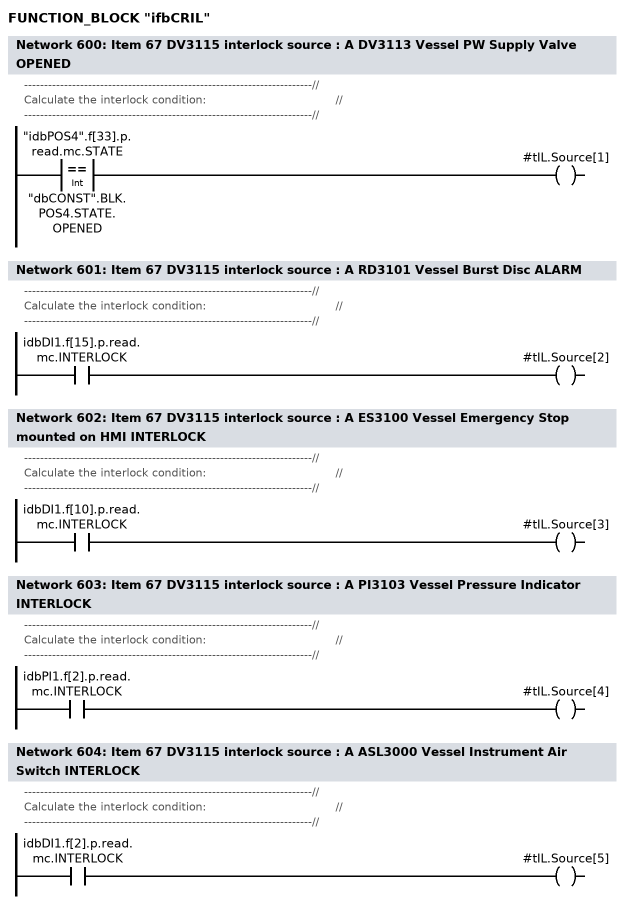
    A(;
    L "idbPOS4".f[33].p.read.mc.STATE;
    L "dbCONST".BLK.POS4.STATE.OPENED;
    ==I;
    );
    = #tIL.Source[1];

NETWORK
TITLE = Item 67 DV3115 interlock source : A RD3101 Vessel Burst Disc ALARM
    //------------------------------------------------------------------------//
    // Calculate the interlock condition:                                     //
    //------------------------------------------------------------------------//
    A idbDI1.f[15].p.read.mc.INTERLOCK;
    = #tIL.Source[2];

NETWORK
TITLE = Item 67 DV3115 interlock source : A ES3100 Vessel Emergency Stop mounted on HMI INTERLOCK
    //------------------------------------------------------------------------//
    // Calculate the interlock condition:                                     //
    //------------------------------------------------------------------------//
    A idbDI1.f[10].p.read.mc.INTERLOCK;
    = #tIL.Source[3];

NETWORK
TITLE = Item 67 DV3115 interlock source : A PI3103 Vessel Pressure Indicator INTERLOCK
    //------------------------------------------------------------------------//
    // Calculate the interlock condition:                                     //
    //------------------------------------------------------------------------//
    A idbPI1.f[2].p.read.mc.INTERLOCK;
    = #tIL.Source[4];

NETWORK
TITLE = Item 67 DV3115 interlock source : A ASL3000 Vessel Instrument Air Switch INTERLOCK
    //------------------------------------------------------------------------//
    // Calculate the interlock condition:                                     //
    //------------------------------------------------------------------------//
    A idbDI1.f[2].p.read.mc.INTERLOCK;
    = #tIL.Source[5];

NETWORK
TITLE = Item 67 DV3115 interlock source : AN ZSC3101 Vessel Manway Closed Indicator CLOSED
    //------------------------------------------------------------------------//
    // Calculate the interlock condition:                                     //
    //------------------------------------------------------------------------//
    AN(;
    L "idbZSC1".f[2].p.read.mc.STATE;
    L "dbCONST".BLK.ZSC1.STATE.CLOSED;
    ==I;
    );
    = #tIL.Source[6];


NETWORK
TITLE = Item 67 DV3115 : Number of interlocks
    //------------------------------------------------------------------------//
    // Number of interlocks
    //------------------------------------------------------------------------//
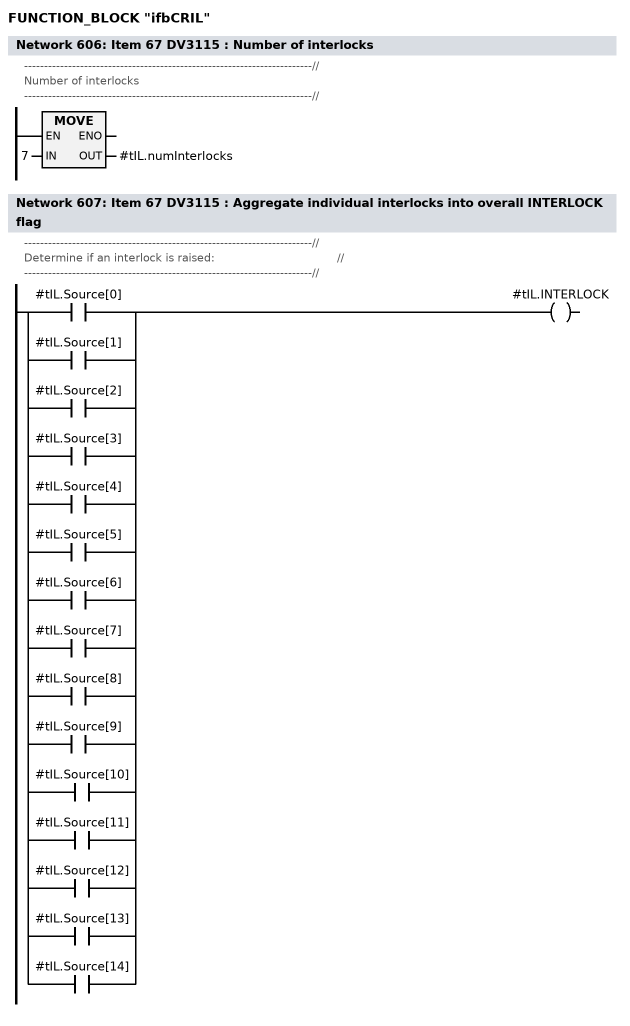
    L 7;
    T #tIL.numInterlocks;

NETWORK
TITLE = Item 67 DV3115 : Aggregate individual interlocks into overall INTERLOCK flag
    //------------------------------------------------------------------------//
    // Determine if an interlock is raised:                                   //
    //------------------------------------------------------------------------//
    O #tIL.Source[0];
    O #tIL.Source[1];
    O #tIL.Source[2];
    O #tIL.Source[3];
    O #tIL.Source[4];
    O #tIL.Source[5];
    O #tIL.Source[6];
    O #tIL.Source[7];
    O #tIL.Source[8];
    O #tIL.Source[9];
    O #tIL.Source[10];
    O #tIL.Source[11];
    O #tIL.Source[12];
    O #tIL.Source[13];
    O #tIL.Source[14];
    = #tIL.INTERLOCK;

NETWORK
TITLE = Item 67 DV3115 : Update the instance data
    //------------------------------------------------------------------------//
    // Update the instance DB with the calculated interlock flags:            //
    //------------------------------------------------------------------------//
    CALL MOVE
    {value_type := 'Variant'}
    (   IN                   := #tIL ,
        OUT                  := #p[67]
    );

NETWORK
TITLE = Item 68 DV3117 : Spray Ball 1 Valve initialise variables
    //------------------------------------------------------------------------//
    // CRITICAL INTERLOCK   CRITICAL INTERLOCK   CRITICAL INTERLOCK   CRITICA //
    // CRITICAL INTERLOCK   CRITICAL INTERLOCK   CRITICAL INTERLOCK   CRITICA //
    //                                                                        //
    // Clear the interlock flag:                                              //
    //------------------------------------------------------------------------//
    A "alwaysLow";
    = #tIL.INTERLOCK;

    //------------------------------------------------------------------------//
    // Clear all interlock values to initialise them to off:                  //
    //------------------------------------------------------------------------//
    CALL FILL_BLK
    {value_type := 'Bool', count_type := 'UInt'}
    (   IN                   := 0 ,
        COUNT                := 15 ,
        OUT                  := #tIL.Source[0]
    );


NETWORK
TITLE = Item 68 DV3117 interlock source : A RD3101 Vessel Burst Disc ALARM
    //------------------------------------------------------------------------//
    // Calculate the interlock condition:                                     //
    //------------------------------------------------------------------------//
    A idbDI1.f[15].p.read.mc.INTERLOCK;
    = #tIL.Source[0];

NETWORK
TITLE = Item 68 DV3117 interlock source : A ES3100 Vessel Emergency Stop mounted on HMI INTERLOCK
    //------------------------------------------------------------------------//
    // Calculate the interlock condition:                                     //
    //------------------------------------------------------------------------//
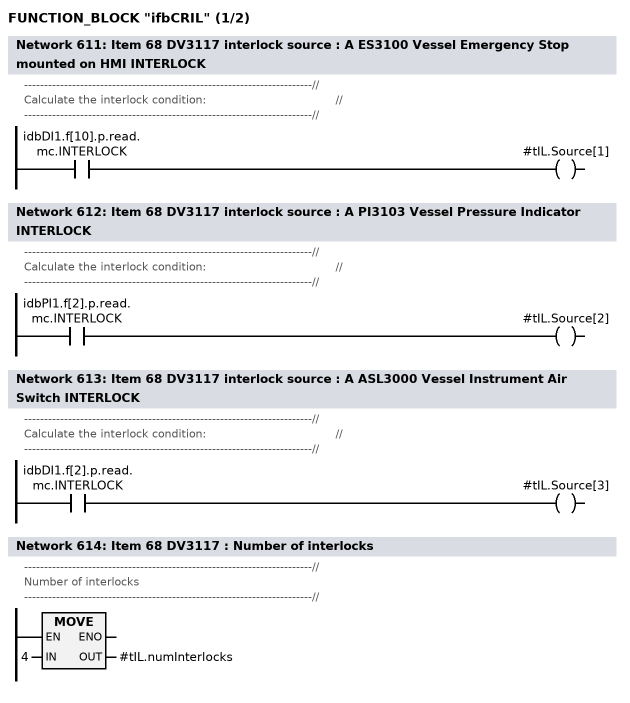
    A idbDI1.f[10].p.read.mc.INTERLOCK;
    = #tIL.Source[1];

NETWORK
TITLE = Item 68 DV3117 interlock source : A PI3103 Vessel Pressure Indicator INTERLOCK
    //------------------------------------------------------------------------//
    // Calculate the interlock condition:                                     //
    //------------------------------------------------------------------------//
    A idbPI1.f[2].p.read.mc.INTERLOCK;
    = #tIL.Source[2];

NETWORK
TITLE = Item 68 DV3117 interlock source : A ASL3000 Vessel Instrument Air Switch INTERLOCK
    //------------------------------------------------------------------------//
    // Calculate the interlock condition:                                     //
    //------------------------------------------------------------------------//
    A idbDI1.f[2].p.read.mc.INTERLOCK;
    = #tIL.Source[3];


NETWORK
TITLE = Item 68 DV3117 : Number of interlocks
    //------------------------------------------------------------------------//
    // Number of interlocks
    //------------------------------------------------------------------------//
    L 4;
    T #tIL.numInterlocks;

NETWORK
TITLE = Item 68 DV3117 : Aggregate individual interlocks into overall INTERLOCK flag
    //------------------------------------------------------------------------//
    // Determine if an interlock is raised:                                   //
    //------------------------------------------------------------------------//
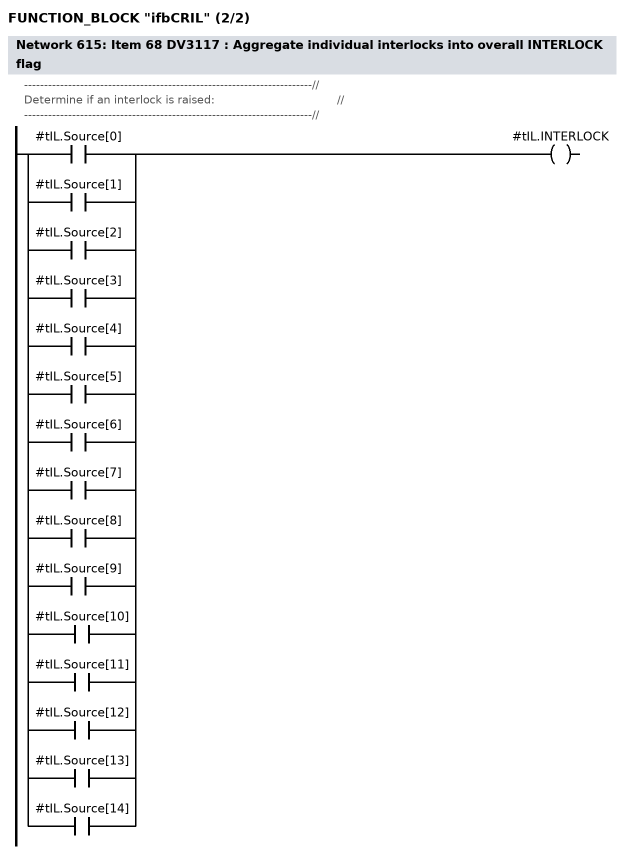
    O #tIL.Source[0];
    O #tIL.Source[1];
    O #tIL.Source[2];
    O #tIL.Source[3];
    O #tIL.Source[4];
    O #tIL.Source[5];
    O #tIL.Source[6];
    O #tIL.Source[7];
    O #tIL.Source[8];
    O #tIL.Source[9];
    O #tIL.Source[10];
    O #tIL.Source[11];
    O #tIL.Source[12];
    O #tIL.Source[13];
    O #tIL.Source[14];
    = #tIL.INTERLOCK;

NETWORK
TITLE = Item 68 DV3117 : Update the instance data
    //------------------------------------------------------------------------//
    // Update the instance DB with the calculated interlock flags:            //
    //------------------------------------------------------------------------//
    CALL MOVE
    {value_type := 'Variant'}
    (   IN                   := #tIL ,
        OUT                  := #p[68]
    );

NETWORK
TITLE = Item 69 DV3119 : Spray Ball 2 Valve initialise variables
    //------------------------------------------------------------------------//
    // CRITICAL INTERLOCK   CRITICAL INTERLOCK   CRITICAL INTERLOCK   CRITICA //
    // CRITICAL INTERLOCK   CRITICAL INTERLOCK   CRITICAL INTERLOCK   CRITICA //
    //                                                                        //
    // Clear the interlock flag:                                              //
    //------------------------------------------------------------------------//
    A "alwaysLow";
    = #tIL.INTERLOCK;

    //------------------------------------------------------------------------//
    // Clear all interlock values to initialise them to off:                  //
    //------------------------------------------------------------------------//
    CALL FILL_BLK
    {value_type := 'Bool', count_type := 'UInt'}
    (   IN                   := 0 ,
        COUNT                := 15 ,
        OUT                  := #tIL.Source[0]
    );


NETWORK
TITLE = Item 69 DV3119 interlock source : A RD3101 Vessel Burst Disc ALARM
    //------------------------------------------------------------------------//
    // Calculate the interlock condition:                                     //
    //------------------------------------------------------------------------//
    A idbDI1.f[15].p.read.mc.INTERLOCK;
    = #tIL.Source[0];

NETWORK
TITLE = Item 69 DV3119 interlock source : A ES3100 Vessel Emergency Stop mounted on HMI INTERLOCK
    //------------------------------------------------------------------------//
    // Calculate the interlock condition:                                     //
    //------------------------------------------------------------------------//
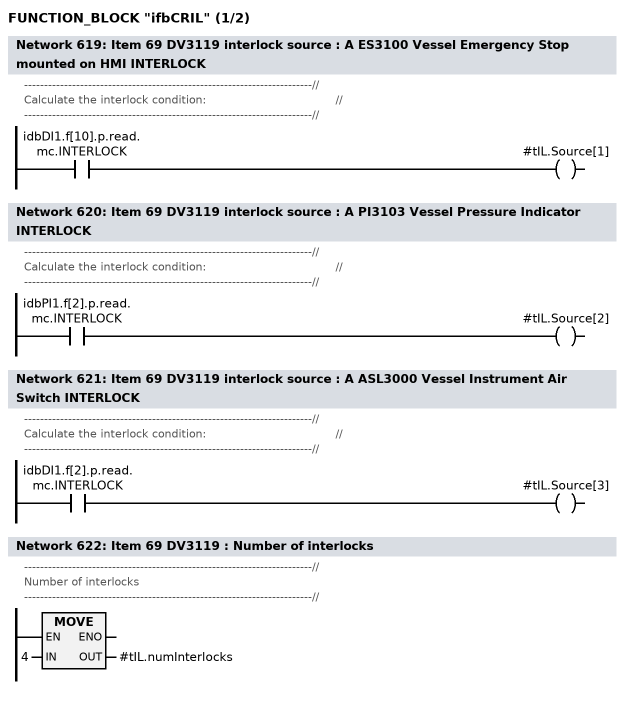
    A idbDI1.f[10].p.read.mc.INTERLOCK;
    = #tIL.Source[1];

NETWORK
TITLE = Item 69 DV3119 interlock source : A PI3103 Vessel Pressure Indicator INTERLOCK
    //------------------------------------------------------------------------//
    // Calculate the interlock condition:                                     //
    //------------------------------------------------------------------------//
    A idbPI1.f[2].p.read.mc.INTERLOCK;
    = #tIL.Source[2];

NETWORK
TITLE = Item 69 DV3119 interlock source : A ASL3000 Vessel Instrument Air Switch INTERLOCK
    //------------------------------------------------------------------------//
    // Calculate the interlock condition:                                     //
    //------------------------------------------------------------------------//
    A idbDI1.f[2].p.read.mc.INTERLOCK;
    = #tIL.Source[3];


NETWORK
TITLE = Item 69 DV3119 : Number of interlocks
    //------------------------------------------------------------------------//
    // Number of interlocks
    //------------------------------------------------------------------------//
    L 4;
    T #tIL.numInterlocks;

NETWORK
TITLE = Item 69 DV3119 : Aggregate individual interlocks into overall INTERLOCK flag
    //------------------------------------------------------------------------//
    // Determine if an interlock is raised:                                   //
    //------------------------------------------------------------------------//
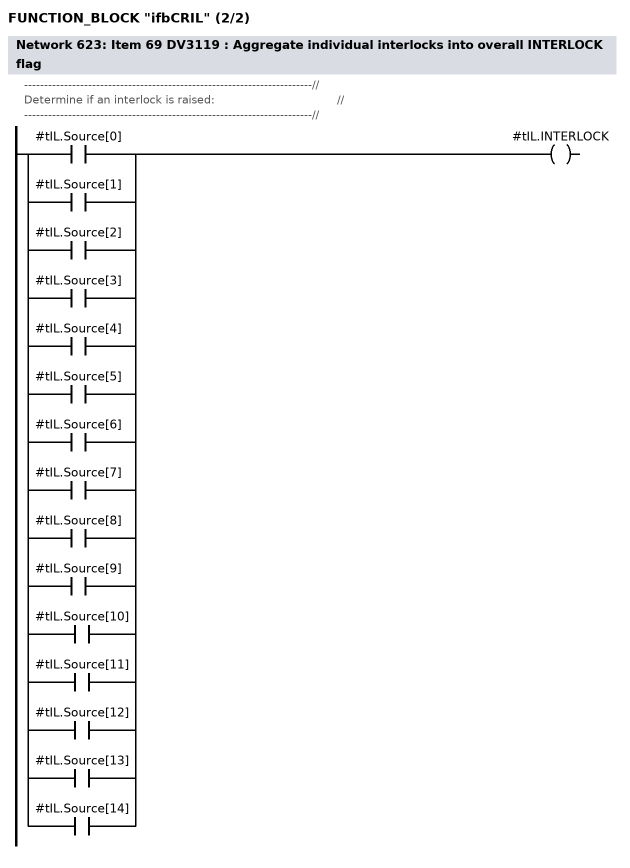
    O #tIL.Source[0];
    O #tIL.Source[1];
    O #tIL.Source[2];
    O #tIL.Source[3];
    O #tIL.Source[4];
    O #tIL.Source[5];
    O #tIL.Source[6];
    O #tIL.Source[7];
    O #tIL.Source[8];
    O #tIL.Source[9];
    O #tIL.Source[10];
    O #tIL.Source[11];
    O #tIL.Source[12];
    O #tIL.Source[13];
    O #tIL.Source[14];
    = #tIL.INTERLOCK;

NETWORK
TITLE = Item 69 DV3119 : Update the instance data
    //------------------------------------------------------------------------//
    // Update the instance DB with the calculated interlock flags:            //
    //------------------------------------------------------------------------//
    CALL MOVE
    {value_type := 'Variant'}
    (   IN                   := #tIL ,
        OUT                  := #p[69]
    );

NETWORK
TITLE = Item 70 DV3121 : Outlet Valve initialise variables
    //------------------------------------------------------------------------//
    // CRITICAL INTERLOCK   CRITICAL INTERLOCK   CRITICAL INTERLOCK   CRITICA //
    // CRITICAL INTERLOCK   CRITICAL INTERLOCK   CRITICAL INTERLOCK   CRITICA //
    //                                                                        //
    // Clear the interlock flag:                                              //
    //------------------------------------------------------------------------//
    A "alwaysLow";
    = #tIL.INTERLOCK;

    //------------------------------------------------------------------------//
    // Clear all interlock values to initialise them to off:                  //
    //------------------------------------------------------------------------//
    CALL FILL_BLK
    {value_type := 'Bool', count_type := 'UInt'}
    (   IN                   := 0 ,
        COUNT                := 15 ,
        OUT                  := #tIL.Source[0]
    );


NETWORK
TITLE = Item 70 DV3121 interlock source : A RD3101 Vessel Burst Disc ALARM
    //------------------------------------------------------------------------//
    // Calculate the interlock condition:                                     //
    //------------------------------------------------------------------------//
    A idbDI1.f[15].p.read.mc.INTERLOCK;
    = #tIL.Source[0];

NETWORK
TITLE = Item 70 DV3121 interlock source : A ES3100 Vessel Emergency Stop mounted on HMI INTERLOCK
    //------------------------------------------------------------------------//
    // Calculate the interlock condition:                                     //
    //------------------------------------------------------------------------//
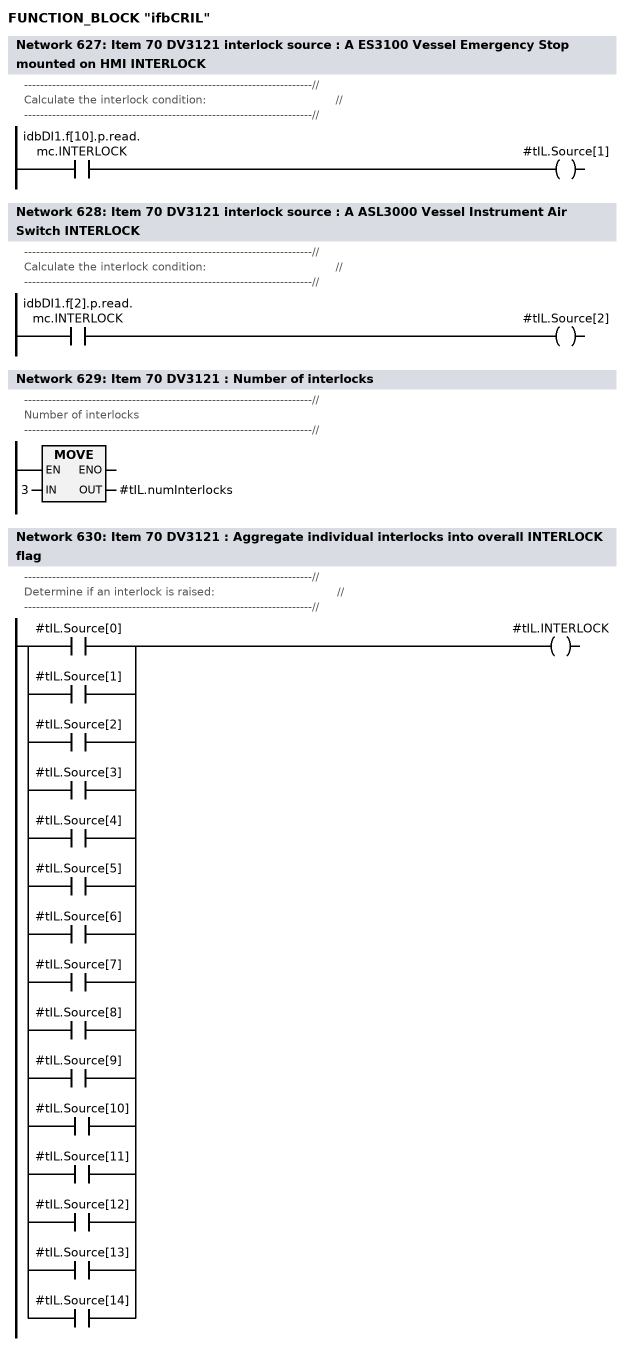
    A idbDI1.f[10].p.read.mc.INTERLOCK;
    = #tIL.Source[1];

NETWORK
TITLE = Item 70 DV3121 interlock source : A ASL3000 Vessel Instrument Air Switch INTERLOCK
    //------------------------------------------------------------------------//
    // Calculate the interlock condition:                                     //
    //------------------------------------------------------------------------//
    A idbDI1.f[2].p.read.mc.INTERLOCK;
    = #tIL.Source[2];


NETWORK
TITLE = Item 70 DV3121 : Number of interlocks
    //------------------------------------------------------------------------//
    // Number of interlocks
    //------------------------------------------------------------------------//
    L 3;
    T #tIL.numInterlocks;

NETWORK
TITLE = Item 70 DV3121 : Aggregate individual interlocks into overall INTERLOCK flag
    //------------------------------------------------------------------------//
    // Determine if an interlock is raised:                                   //
    //------------------------------------------------------------------------//
    O #tIL.Source[0];
    O #tIL.Source[1];
    O #tIL.Source[2];
    O #tIL.Source[3];
    O #tIL.Source[4];
    O #tIL.Source[5];
    O #tIL.Source[6];
    O #tIL.Source[7];
    O #tIL.Source[8];
    O #tIL.Source[9];
    O #tIL.Source[10];
    O #tIL.Source[11];
    O #tIL.Source[12];
    O #tIL.Source[13];
    O #tIL.Source[14];
    = #tIL.INTERLOCK;

NETWORK
TITLE = Item 70 DV3121 : Update the instance data
    //------------------------------------------------------------------------//
    // Update the instance DB with the calculated interlock flags:            //
    //------------------------------------------------------------------------//
    CALL MOVE
    {value_type := 'Variant'}
    (   IN                   := #tIL ,
        OUT                  := #p[70]
    );

NETWORK
TITLE = Item 71 DV3125 : Sy Transfer line Valve Matrix SMFLx initialise variables
    //------------------------------------------------------------------------//
    // CRITICAL INTERLOCK   CRITICAL INTERLOCK   CRITICAL INTERLOCK   CRITICA //
    // CRITICAL INTERLOCK   CRITICAL INTERLOCK   CRITICAL INTERLOCK   CRITICA //
    //                                                                        //
    // Clear the interlock flag:                                              //
    //------------------------------------------------------------------------//
    A "alwaysLow";
    = #tIL.INTERLOCK;

    //------------------------------------------------------------------------//
    // Clear all interlock values to initialise them to off:                  //
    //------------------------------------------------------------------------//
    CALL FILL_BLK
    {value_type := 'Bool', count_type := 'UInt'}
    (   IN                   := 0 ,
        COUNT                := 15 ,
        OUT                  := #tIL.Source[0]
    );


NETWORK
TITLE = Item 71 DV3125 interlock source : AN ZSC3111 SMFL1 to S1/BFS1 Flowpath Indicator IN   AN ZSC3113 SMFL2 to S1/BFS1 Flowpath Indicator IN
    //------------------------------------------------------------------------//
    // Calculate the interlock condition:                                     //
    //------------------------------------------------------------------------//
    AN(;
    L "idbZSC2".f[17].p.read.mc.STATE;
    L "dbCONST".BLK.ZSC2.STATE.IN;
    ==I;
    );
AN(;
    L "idbZSC2".f[18].p.read.mc.STATE;
    L "dbCONST".BLK.ZSC2.STATE.IN;
    ==I;
    );
    = #tIL.Source[0];


NETWORK
TITLE = Item 71 DV3125 : Number of interlocks
    //------------------------------------------------------------------------//
    // Number of interlocks
    //------------------------------------------------------------------------//
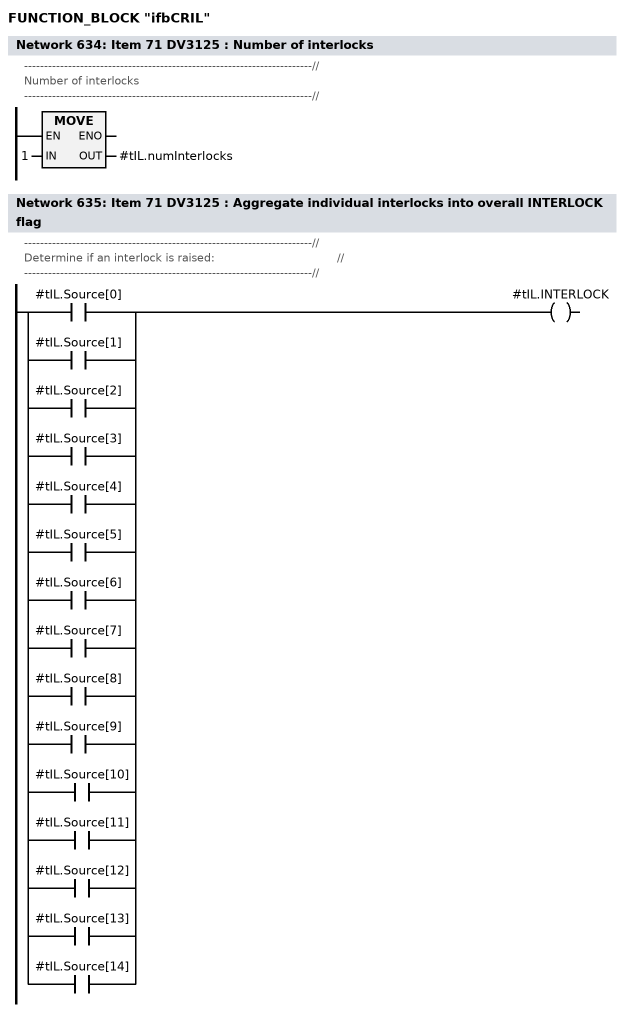
    L 1;
    T #tIL.numInterlocks;

NETWORK
TITLE = Item 71 DV3125 : Aggregate individual interlocks into overall INTERLOCK flag
    //------------------------------------------------------------------------//
    // Determine if an interlock is raised:                                   //
    //------------------------------------------------------------------------//
    O #tIL.Source[0];
    O #tIL.Source[1];
    O #tIL.Source[2];
    O #tIL.Source[3];
    O #tIL.Source[4];
    O #tIL.Source[5];
    O #tIL.Source[6];
    O #tIL.Source[7];
    O #tIL.Source[8];
    O #tIL.Source[9];
    O #tIL.Source[10];
    O #tIL.Source[11];
    O #tIL.Source[12];
    O #tIL.Source[13];
    O #tIL.Source[14];
    = #tIL.INTERLOCK;

NETWORK
TITLE = Item 71 DV3125 : Update the instance data
    //------------------------------------------------------------------------//
    // Update the instance DB with the calculated interlock flags:            //
    //------------------------------------------------------------------------//
    CALL MOVE
    {value_type := 'Variant'}
    (   IN                   := #tIL ,
        OUT                  := #p[71]
    );

NETWORK
TITLE = Item 72 DV3129 : Sy Transfer line Valve Matrix FLz initialise variables
    //------------------------------------------------------------------------//
    // CRITICAL INTERLOCK   CRITICAL INTERLOCK   CRITICAL INTERLOCK   CRITICA //
    // CRITICAL INTERLOCK   CRITICAL INTERLOCK   CRITICAL INTERLOCK   CRITICA //
    //                                                                        //
    // Clear the interlock flag:                                              //
    //------------------------------------------------------------------------//
    A "alwaysLow";
    = #tIL.INTERLOCK;

    //------------------------------------------------------------------------//
    // Clear all interlock values to initialise them to off:                  //
    //------------------------------------------------------------------------//
    CALL FILL_BLK
    {value_type := 'Bool', count_type := 'UInt'}
    (   IN                   := 0 ,
        COUNT                := 15 ,
        OUT                  := #tIL.Source[0]
    );


NETWORK
TITLE = Item 72 DV3129 interlock source : AN ZSC3115 S1 to F1P1 Flowpath Indicator IN   AN ZSC3117 S1 to F2P1 Flowpath Indicator IN
    //------------------------------------------------------------------------//
    // Calculate the interlock condition:                                     //
    //------------------------------------------------------------------------//
    AN(;
    L "idbZSC2".f[19].p.read.mc.STATE;
    L "dbCONST".BLK.ZSC2.STATE.IN;
    ==I;
    );
AN(;
    L "idbZSC2".f[20].p.read.mc.STATE;
    L "dbCONST".BLK.ZSC2.STATE.IN;
    ==I;
    );
    = #tIL.Source[0];


NETWORK
TITLE = Item 72 DV3129 : Number of interlocks
    //------------------------------------------------------------------------//
    // Number of interlocks
    //------------------------------------------------------------------------//
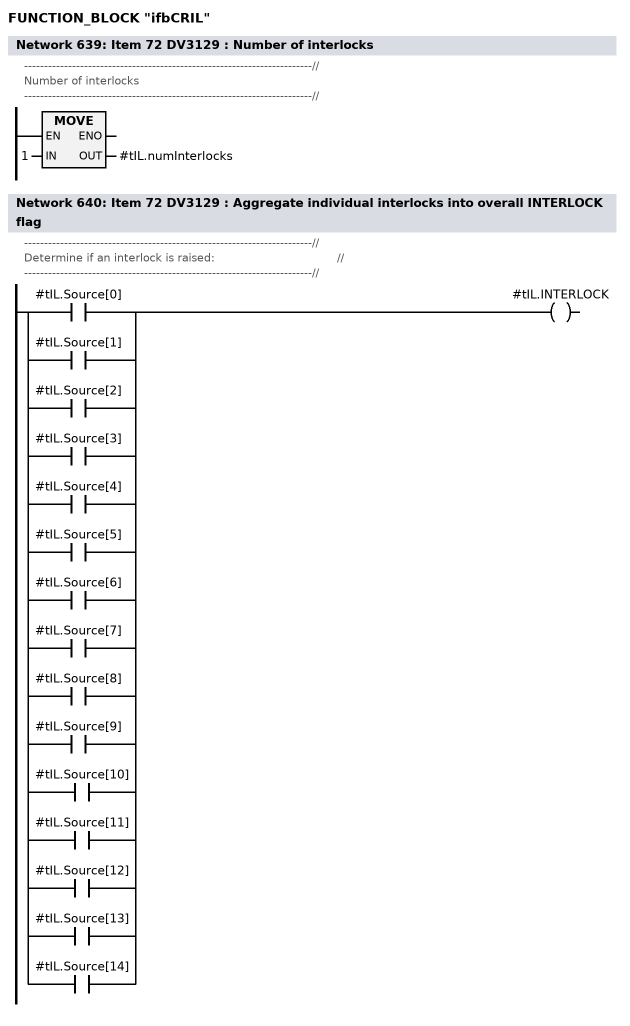
    L 1;
    T #tIL.numInterlocks;

NETWORK
TITLE = Item 72 DV3129 : Aggregate individual interlocks into overall INTERLOCK flag
    //------------------------------------------------------------------------//
    // Determine if an interlock is raised:                                   //
    //------------------------------------------------------------------------//
    O #tIL.Source[0];
    O #tIL.Source[1];
    O #tIL.Source[2];
    O #tIL.Source[3];
    O #tIL.Source[4];
    O #tIL.Source[5];
    O #tIL.Source[6];
    O #tIL.Source[7];
    O #tIL.Source[8];
    O #tIL.Source[9];
    O #tIL.Source[10];
    O #tIL.Source[11];
    O #tIL.Source[12];
    O #tIL.Source[13];
    O #tIL.Source[14];
    = #tIL.INTERLOCK;

NETWORK
TITLE = Item 72 DV3129 : Update the instance data
    //------------------------------------------------------------------------//
    // Update the instance DB with the calculated interlock flags:            //
    //------------------------------------------------------------------------//
    CALL MOVE
    {value_type := 'Variant'}
    (   IN                   := #tIL ,
        OUT                  := #p[72]
    );

NETWORK
TITLE = Item 73 DV4101 : Vent Valve initialise variables
    //------------------------------------------------------------------------//
    // CRITICAL INTERLOCK   CRITICAL INTERLOCK   CRITICAL INTERLOCK   CRITICA //
    // CRITICAL INTERLOCK   CRITICAL INTERLOCK   CRITICAL INTERLOCK   CRITICA //
    //                                                                        //
    // Clear the interlock flag:                                              //
    //------------------------------------------------------------------------//
    A "alwaysLow";
    = #tIL.INTERLOCK;

    //------------------------------------------------------------------------//
    // Clear all interlock values to initialise them to off:                  //
    //------------------------------------------------------------------------//
    CALL FILL_BLK
    {value_type := 'Bool', count_type := 'UInt'}
    (   IN                   := 0 ,
        COUNT                := 15 ,
        OUT                  := #tIL.Source[0]
    );


NETWORK
TITLE = Item 73 DV4101 interlock source : A RD4101 Vessel Burst Disc ALARM
    //------------------------------------------------------------------------//
    // Calculate the interlock condition:                                     //
    //------------------------------------------------------------------------//
    A idbDI1.f[16].p.read.mc.INTERLOCK;
    = #tIL.Source[0];

NETWORK
TITLE = Item 73 DV4101 interlock source : A ES4100 Vessel Emergency Stop mounted on HMI INTERLOCK
    //------------------------------------------------------------------------//
    // Calculate the interlock condition:                                     //
    //------------------------------------------------------------------------//
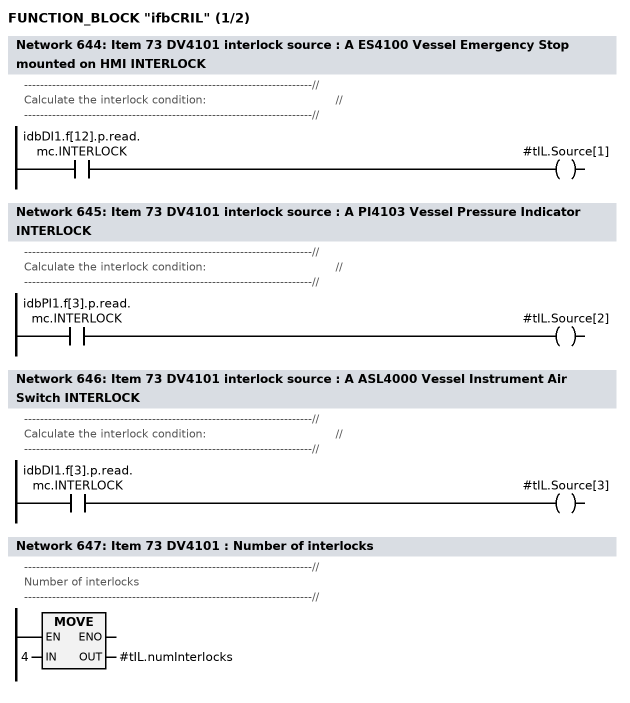
    A idbDI1.f[12].p.read.mc.INTERLOCK;
    = #tIL.Source[1];

NETWORK
TITLE = Item 73 DV4101 interlock source : A PI4103 Vessel Pressure Indicator INTERLOCK
    //------------------------------------------------------------------------//
    // Calculate the interlock condition:                                     //
    //------------------------------------------------------------------------//
    A idbPI1.f[3].p.read.mc.INTERLOCK;
    = #tIL.Source[2];

NETWORK
TITLE = Item 73 DV4101 interlock source : A ASL4000 Vessel Instrument Air Switch INTERLOCK
    //------------------------------------------------------------------------//
    // Calculate the interlock condition:                                     //
    //------------------------------------------------------------------------//
    A idbDI1.f[3].p.read.mc.INTERLOCK;
    = #tIL.Source[3];


NETWORK
TITLE = Item 73 DV4101 : Number of interlocks
    //------------------------------------------------------------------------//
    // Number of interlocks
    //------------------------------------------------------------------------//
    L 4;
    T #tIL.numInterlocks;

NETWORK
TITLE = Item 73 DV4101 : Aggregate individual interlocks into overall INTERLOCK flag
    //------------------------------------------------------------------------//
    // Determine if an interlock is raised:                                   //
    //------------------------------------------------------------------------//
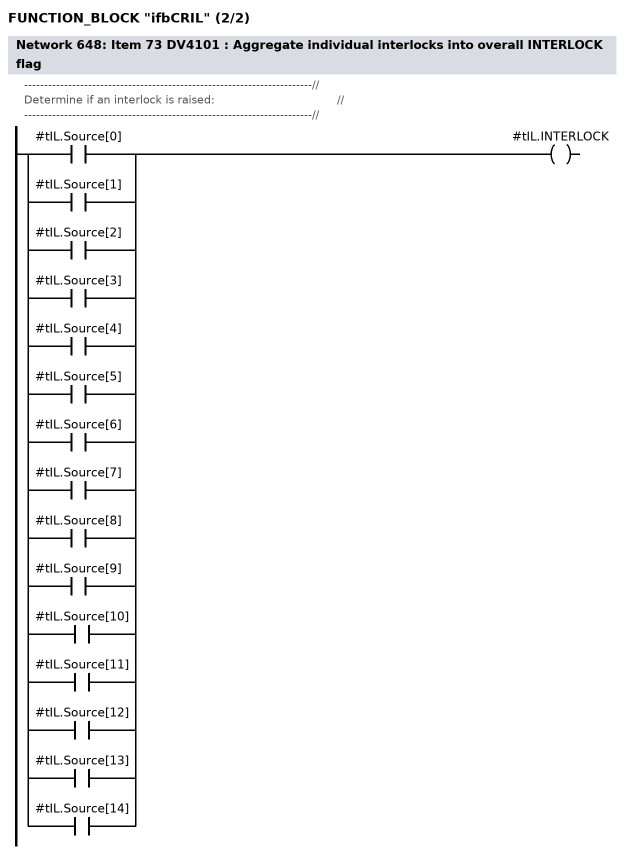
    O #tIL.Source[0];
    O #tIL.Source[1];
    O #tIL.Source[2];
    O #tIL.Source[3];
    O #tIL.Source[4];
    O #tIL.Source[5];
    O #tIL.Source[6];
    O #tIL.Source[7];
    O #tIL.Source[8];
    O #tIL.Source[9];
    O #tIL.Source[10];
    O #tIL.Source[11];
    O #tIL.Source[12];
    O #tIL.Source[13];
    O #tIL.Source[14];
    = #tIL.INTERLOCK;

NETWORK
TITLE = Item 73 DV4101 : Update the instance data
    //------------------------------------------------------------------------//
    // Update the instance DB with the calculated interlock flags:            //
    //------------------------------------------------------------------------//
    CALL MOVE
    {value_type := 'Variant'}
    (   IN                   := #tIL ,
        OUT                  := #p[73]
    );

NETWORK
TITLE = Item 74 DV4103 : HP CA Supply Valve initialise variables
    //------------------------------------------------------------------------//
    // CRITICAL INTERLOCK   CRITICAL INTERLOCK   CRITICAL INTERLOCK   CRITICA //
    // CRITICAL INTERLOCK   CRITICAL INTERLOCK   CRITICAL INTERLOCK   CRITICA //
    //                                                                        //
    // Clear the interlock flag:                                              //
    //------------------------------------------------------------------------//
    A "alwaysLow";
    = #tIL.INTERLOCK;

    //------------------------------------------------------------------------//
    // Clear all interlock values to initialise them to off:                  //
    //------------------------------------------------------------------------//
    CALL FILL_BLK
    {value_type := 'Bool', count_type := 'UInt'}
    (   IN                   := 0 ,
        COUNT                := 15 ,
        OUT                  := #tIL.Source[0]
    );


NETWORK
TITLE = Item 74 DV4103 interlock source : A RD4101 Vessel Burst Disc ALARM
    //------------------------------------------------------------------------//
    // Calculate the interlock condition:                                     //
    //------------------------------------------------------------------------//
    A idbDI1.f[16].p.read.mc.INTERLOCK;
    = #tIL.Source[0];

NETWORK
TITLE = Item 74 DV4103 interlock source : A ES4100 Vessel Emergency Stop mounted on HMI INTERLOCK
    //------------------------------------------------------------------------//
    // Calculate the interlock condition:                                     //
    //------------------------------------------------------------------------//
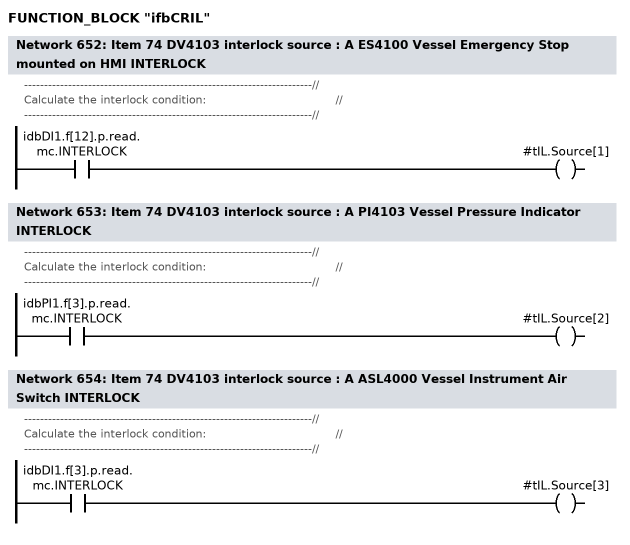
    A idbDI1.f[12].p.read.mc.INTERLOCK;
    = #tIL.Source[1];

NETWORK
TITLE = Item 74 DV4103 interlock source : A PI4103 Vessel Pressure Indicator INTERLOCK
    //------------------------------------------------------------------------//
    // Calculate the interlock condition:                                     //
    //------------------------------------------------------------------------//
    A idbPI1.f[3].p.read.mc.INTERLOCK;
    = #tIL.Source[2];

NETWORK
TITLE = Item 74 DV4103 interlock source : A ASL4000 Vessel Instrument Air Switch INTERLOCK
    //------------------------------------------------------------------------//
    // Calculate the interlock condition:                                     //
    //------------------------------------------------------------------------//
    A idbDI1.f[3].p.read.mc.INTERLOCK;
    = #tIL.Source[3];

NETWORK
TITLE = Item 74 DV4103 interlock source : AN ZSC4101 Vessel Manway Closed Indicator CLOSED
    //------------------------------------------------------------------------//
    // Calculate the interlock condition:                                     //
    //------------------------------------------------------------------------//
    AN(;
    L "idbZSC1".f[3].p.read.mc.STATE;
    L "dbCONST".BLK.ZSC1.STATE.CLOSED;
    ==I;
    );
    = #tIL.Source[4];


NETWORK
TITLE = Item 74 DV4103 : Number of interlocks
    //------------------------------------------------------------------------//
    // Number of interlocks
    //------------------------------------------------------------------------//
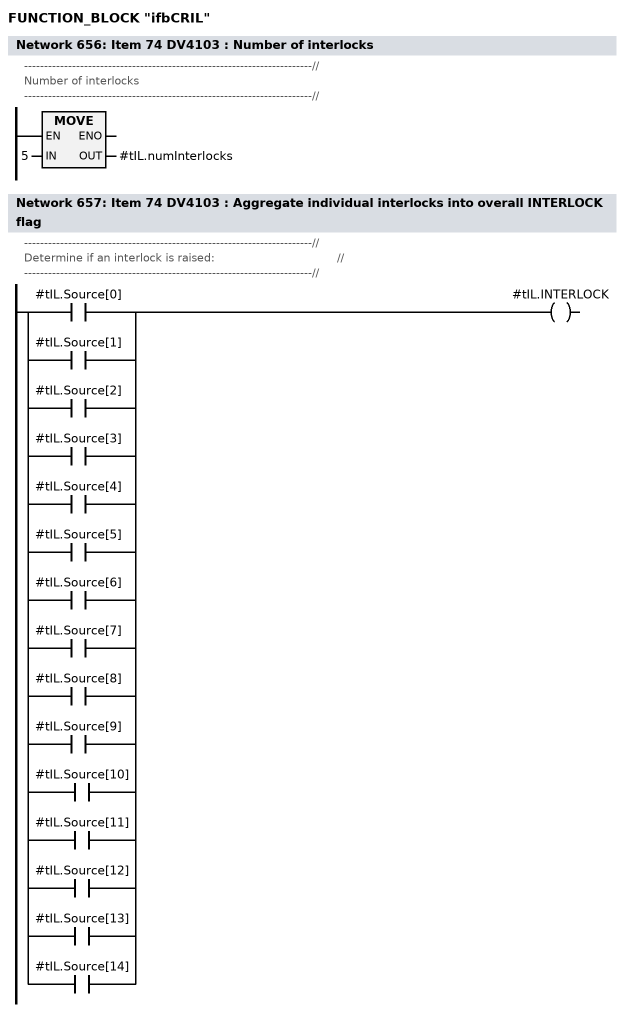
    L 5;
    T #tIL.numInterlocks;

NETWORK
TITLE = Item 74 DV4103 : Aggregate individual interlocks into overall INTERLOCK flag
    //------------------------------------------------------------------------//
    // Determine if an interlock is raised:                                   //
    //------------------------------------------------------------------------//
    O #tIL.Source[0];
    O #tIL.Source[1];
    O #tIL.Source[2];
    O #tIL.Source[3];
    O #tIL.Source[4];
    O #tIL.Source[5];
    O #tIL.Source[6];
    O #tIL.Source[7];
    O #tIL.Source[8];
    O #tIL.Source[9];
    O #tIL.Source[10];
    O #tIL.Source[11];
    O #tIL.Source[12];
    O #tIL.Source[13];
    O #tIL.Source[14];
    = #tIL.INTERLOCK;

NETWORK
TITLE = Item 74 DV4103 : Update the instance data
    //------------------------------------------------------------------------//
    // Update the instance DB with the calculated interlock flags:            //
    //------------------------------------------------------------------------//
    CALL MOVE
    {value_type := 'Variant'}
    (   IN                   := #tIL ,
        OUT                  := #p[74]
    );

NETWORK
TITLE = Item 75 DV4105 : LP CA Supply Valve initialise variables
    //------------------------------------------------------------------------//
    // CRITICAL INTERLOCK   CRITICAL INTERLOCK   CRITICAL INTERLOCK   CRITICA //
    // CRITICAL INTERLOCK   CRITICAL INTERLOCK   CRITICAL INTERLOCK   CRITICA //
    //                                                                        //
    // Clear the interlock flag:                                              //
    //------------------------------------------------------------------------//
    A "alwaysLow";
    = #tIL.INTERLOCK;

    //------------------------------------------------------------------------//
    // Clear all interlock values to initialise them to off:                  //
    //------------------------------------------------------------------------//
    CALL FILL_BLK
    {value_type := 'Bool', count_type := 'UInt'}
    (   IN                   := 0 ,
        COUNT                := 15 ,
        OUT                  := #tIL.Source[0]
    );


NETWORK
TITLE = Item 75 DV4105 interlock source : A RD4101 Vessel Burst Disc ALARM
    //------------------------------------------------------------------------//
    // Calculate the interlock condition:                                     //
    //------------------------------------------------------------------------//
    A idbDI1.f[16].p.read.mc.INTERLOCK;
    = #tIL.Source[0];

NETWORK
TITLE = Item 75 DV4105 interlock source : A ES4100 Vessel Emergency Stop mounted on HMI INTERLOCK
    //------------------------------------------------------------------------//
    // Calculate the interlock condition:                                     //
    //------------------------------------------------------------------------//
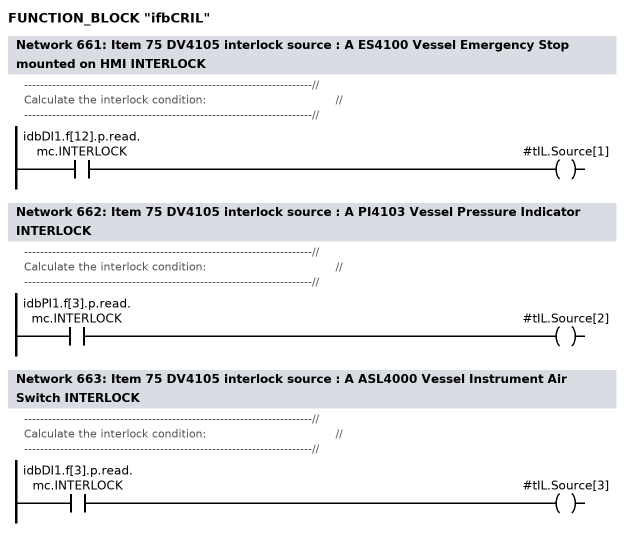
    A idbDI1.f[12].p.read.mc.INTERLOCK;
    = #tIL.Source[1];

NETWORK
TITLE = Item 75 DV4105 interlock source : A PI4103 Vessel Pressure Indicator INTERLOCK
    //------------------------------------------------------------------------//
    // Calculate the interlock condition:                                     //
    //------------------------------------------------------------------------//
    A idbPI1.f[3].p.read.mc.INTERLOCK;
    = #tIL.Source[2];

NETWORK
TITLE = Item 75 DV4105 interlock source : A ASL4000 Vessel Instrument Air Switch INTERLOCK
    //------------------------------------------------------------------------//
    // Calculate the interlock condition:                                     //
    //------------------------------------------------------------------------//
    A idbDI1.f[3].p.read.mc.INTERLOCK;
    = #tIL.Source[3];

NETWORK
TITLE = Item 75 DV4105 interlock source : AN ZSC4101 Vessel Manway Closed Indicator CLOSED
    //------------------------------------------------------------------------//
    // Calculate the interlock condition:                                     //
    //------------------------------------------------------------------------//
    AN(;
    L "idbZSC1".f[3].p.read.mc.STATE;
    L "dbCONST".BLK.ZSC1.STATE.CLOSED;
    ==I;
    );
    = #tIL.Source[4];


NETWORK
TITLE = Item 75 DV4105 : Number of interlocks
    //------------------------------------------------------------------------//
    // Number of interlocks
    //------------------------------------------------------------------------//
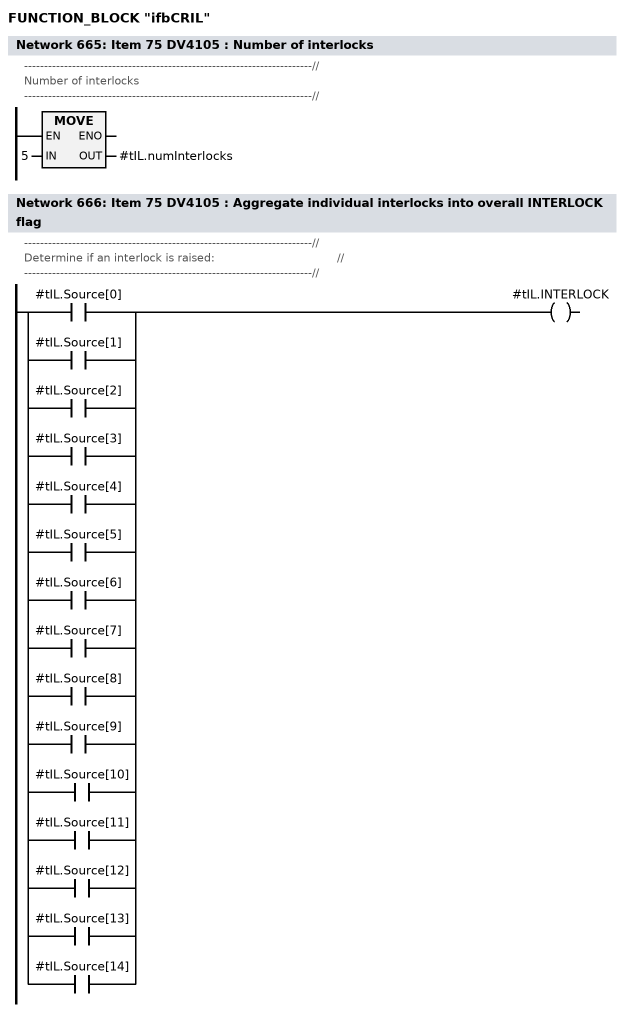
    L 5;
    T #tIL.numInterlocks;

NETWORK
TITLE = Item 75 DV4105 : Aggregate individual interlocks into overall INTERLOCK flag
    //------------------------------------------------------------------------//
    // Determine if an interlock is raised:                                   //
    //------------------------------------------------------------------------//
    O #tIL.Source[0];
    O #tIL.Source[1];
    O #tIL.Source[2];
    O #tIL.Source[3];
    O #tIL.Source[4];
    O #tIL.Source[5];
    O #tIL.Source[6];
    O #tIL.Source[7];
    O #tIL.Source[8];
    O #tIL.Source[9];
    O #tIL.Source[10];
    O #tIL.Source[11];
    O #tIL.Source[12];
    O #tIL.Source[13];
    O #tIL.Source[14];
    = #tIL.INTERLOCK;

NETWORK
TITLE = Item 75 DV4105 : Update the instance data
    //------------------------------------------------------------------------//
    // Update the instance DB with the calculated interlock flags:            //
    //------------------------------------------------------------------------//
    CALL MOVE
    {value_type := 'Variant'}
    (   IN                   := #tIL ,
        OUT                  := #p[75]
    );

NETWORK
TITLE = Item 76 DV4107 : Vacuum valve initialise variables
    //------------------------------------------------------------------------//
    // CRITICAL INTERLOCK   CRITICAL INTERLOCK   CRITICAL INTERLOCK   CRITICA //
    // CRITICAL INTERLOCK   CRITICAL INTERLOCK   CRITICAL INTERLOCK   CRITICA //
    //                                                                        //
    // Clear the interlock flag:                                              //
    //------------------------------------------------------------------------//
    A "alwaysLow";
    = #tIL.INTERLOCK;

    //------------------------------------------------------------------------//
    // Clear all interlock values to initialise them to off:                  //
    //------------------------------------------------------------------------//
    CALL FILL_BLK
    {value_type := 'Bool', count_type := 'UInt'}
    (   IN                   := 0 ,
        COUNT                := 15 ,
        OUT                  := #tIL.Source[0]
    );


NETWORK
TITLE = Item 76 DV4107 interlock source : A RD4101 Vessel Burst Disc ALARM
    //------------------------------------------------------------------------//
    // Calculate the interlock condition:                                     //
    //------------------------------------------------------------------------//
    A idbDI1.f[16].p.read.mc.INTERLOCK;
    = #tIL.Source[0];

NETWORK
TITLE = Item 76 DV4107 interlock source : A ES4100 Vessel Emergency Stop mounted on HMI INTERLOCK
    //------------------------------------------------------------------------//
    // Calculate the interlock condition:                                     //
    //------------------------------------------------------------------------//
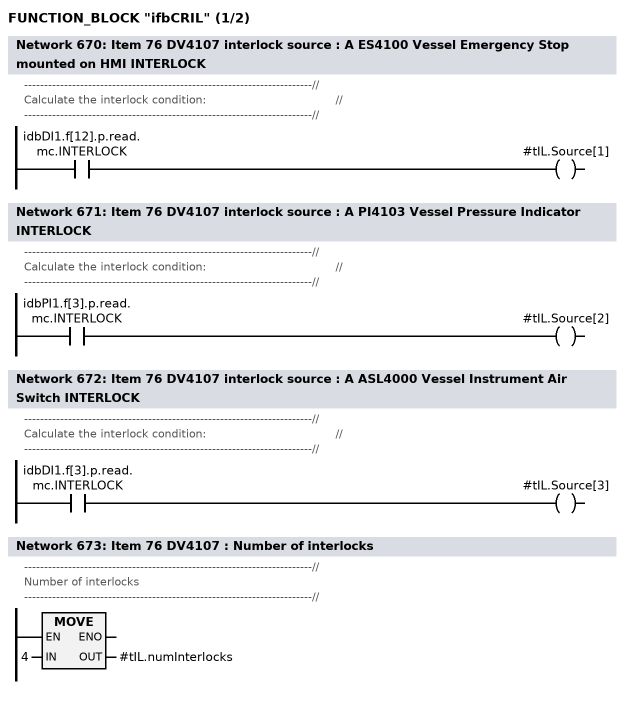
    A idbDI1.f[12].p.read.mc.INTERLOCK;
    = #tIL.Source[1];

NETWORK
TITLE = Item 76 DV4107 interlock source : A PI4103 Vessel Pressure Indicator INTERLOCK
    //------------------------------------------------------------------------//
    // Calculate the interlock condition:                                     //
    //------------------------------------------------------------------------//
    A idbPI1.f[3].p.read.mc.INTERLOCK;
    = #tIL.Source[2];

NETWORK
TITLE = Item 76 DV4107 interlock source : A ASL4000 Vessel Instrument Air Switch INTERLOCK
    //------------------------------------------------------------------------//
    // Calculate the interlock condition:                                     //
    //------------------------------------------------------------------------//
    A idbDI1.f[3].p.read.mc.INTERLOCK;
    = #tIL.Source[3];


NETWORK
TITLE = Item 76 DV4107 : Number of interlocks
    //------------------------------------------------------------------------//
    // Number of interlocks
    //------------------------------------------------------------------------//
    L 4;
    T #tIL.numInterlocks;

NETWORK
TITLE = Item 76 DV4107 : Aggregate individual interlocks into overall INTERLOCK flag
    //------------------------------------------------------------------------//
    // Determine if an interlock is raised:                                   //
    //------------------------------------------------------------------------//
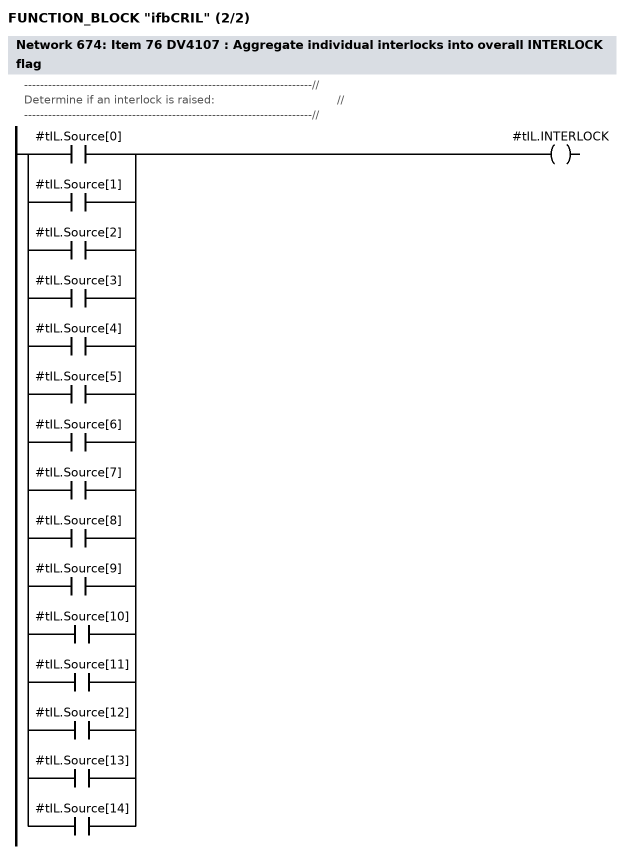
    O #tIL.Source[0];
    O #tIL.Source[1];
    O #tIL.Source[2];
    O #tIL.Source[3];
    O #tIL.Source[4];
    O #tIL.Source[5];
    O #tIL.Source[6];
    O #tIL.Source[7];
    O #tIL.Source[8];
    O #tIL.Source[9];
    O #tIL.Source[10];
    O #tIL.Source[11];
    O #tIL.Source[12];
    O #tIL.Source[13];
    O #tIL.Source[14];
    = #tIL.INTERLOCK;

NETWORK
TITLE = Item 76 DV4107 : Update the instance data
    //------------------------------------------------------------------------//
    // Update the instance DB with the calculated interlock flags:            //
    //------------------------------------------------------------------------//
    CALL MOVE
    {value_type := 'Variant'}
    (   IN                   := #tIL ,
        OUT                  := #p[76]
    );

NETWORK
TITLE = Item 77 DV4109 : PS Supply for WFI Loop initialise variables
    //------------------------------------------------------------------------//
    // CRITICAL INTERLOCK   CRITICAL INTERLOCK   CRITICAL INTERLOCK   CRITICA //
    // CRITICAL INTERLOCK   CRITICAL INTERLOCK   CRITICAL INTERLOCK   CRITICA //
    //                                                                        //
    // Clear the interlock flag:                                              //
    //------------------------------------------------------------------------//
    A "alwaysLow";
    = #tIL.INTERLOCK;

    //------------------------------------------------------------------------//
    // Clear all interlock values to initialise them to off:                  //
    //------------------------------------------------------------------------//
    CALL FILL_BLK
    {value_type := 'Bool', count_type := 'UInt'}
    (   IN                   := 0 ,
        COUNT                := 15 ,
        OUT                  := #tIL.Source[0]
    );


NETWORK
TITLE = Item 77 DV4109 interlock source : ON ZSC4107 Vessel inlet line Flowpath Indicator IN   ON ZSC4103 Vessel WFI Supply Flowpath Indicator IN
    //------------------------------------------------------------------------//
    // Calculate the interlock condition:                                     //
    //------------------------------------------------------------------------//
    ON(;
    L "idbZSC2".f[23].p.read.mc.STATE;
    L "dbCONST".BLK.ZSC2.STATE.IN;
    ==I;
    );
ON(;
    L "idbZSC2".f[21].p.read.mc.STATE;
    L "dbCONST".BLK.ZSC2.STATE.IN;
    ==I;
    );
    = #tIL.Source[0];

NETWORK
TITLE = Item 77 DV4109 interlock source : A DV4111 Vessel WFI Supply Valve OPENED
    //------------------------------------------------------------------------//
    // Calculate the interlock condition:                                     //
    //------------------------------------------------------------------------//
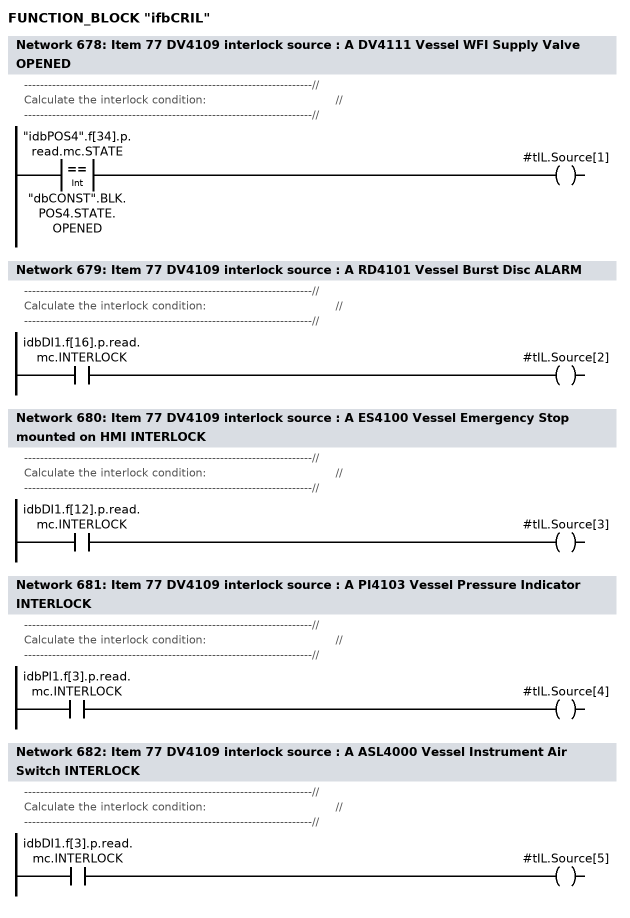
    A(;
    L "idbPOS4".f[34].p.read.mc.STATE;
    L "dbCONST".BLK.POS4.STATE.OPENED;
    ==I;
    );
    = #tIL.Source[1];

NETWORK
TITLE = Item 77 DV4109 interlock source : A RD4101 Vessel Burst Disc ALARM
    //------------------------------------------------------------------------//
    // Calculate the interlock condition:                                     //
    //------------------------------------------------------------------------//
    A idbDI1.f[16].p.read.mc.INTERLOCK;
    = #tIL.Source[2];

NETWORK
TITLE = Item 77 DV4109 interlock source : A ES4100 Vessel Emergency Stop mounted on HMI INTERLOCK
    //------------------------------------------------------------------------//
    // Calculate the interlock condition:                                     //
    //------------------------------------------------------------------------//
    A idbDI1.f[12].p.read.mc.INTERLOCK;
    = #tIL.Source[3];

NETWORK
TITLE = Item 77 DV4109 interlock source : A PI4103 Vessel Pressure Indicator INTERLOCK
    //------------------------------------------------------------------------//
    // Calculate the interlock condition:                                     //
    //------------------------------------------------------------------------//
    A idbPI1.f[3].p.read.mc.INTERLOCK;
    = #tIL.Source[4];

NETWORK
TITLE = Item 77 DV4109 interlock source : A ASL4000 Vessel Instrument Air Switch INTERLOCK
    //------------------------------------------------------------------------//
    // Calculate the interlock condition:                                     //
    //------------------------------------------------------------------------//
    A idbDI1.f[3].p.read.mc.INTERLOCK;
    = #tIL.Source[5];

NETWORK
TITLE = Item 77 DV4109 interlock source : AN ZSC4101 Vessel Manway Closed Indicator CLOSED
    //------------------------------------------------------------------------//
    // Calculate the interlock condition:                                     //
    //------------------------------------------------------------------------//
    AN(;
    L "idbZSC1".f[3].p.read.mc.STATE;
    L "dbCONST".BLK.ZSC1.STATE.CLOSED;
    ==I;
    );
    = #tIL.Source[6];


NETWORK
TITLE = Item 77 DV4109 : Number of interlocks
    //------------------------------------------------------------------------//
    // Number of interlocks
    //------------------------------------------------------------------------//
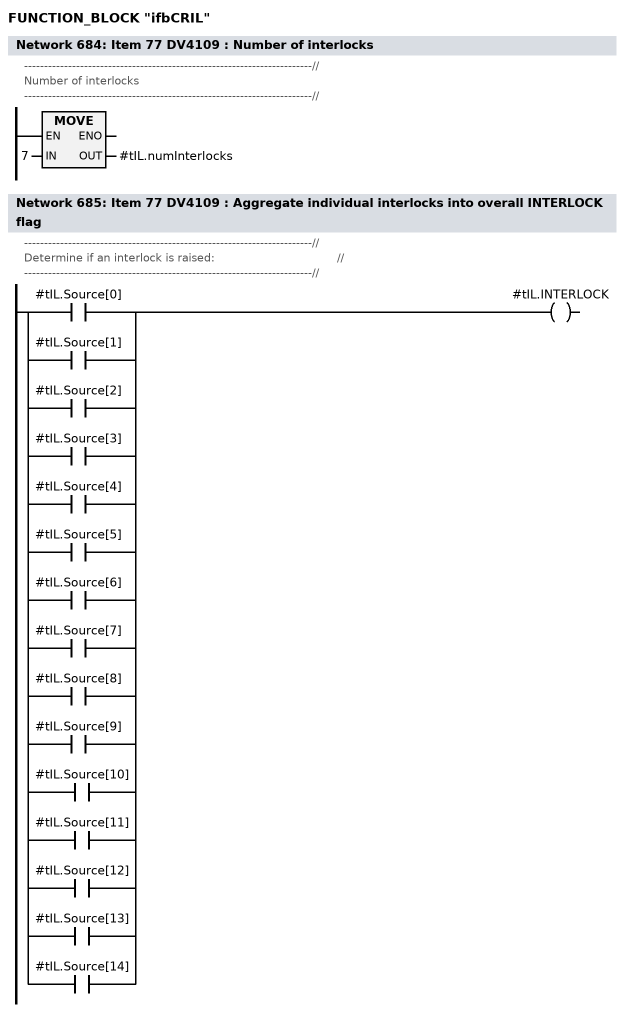
    L 7;
    T #tIL.numInterlocks;

NETWORK
TITLE = Item 77 DV4109 : Aggregate individual interlocks into overall INTERLOCK flag
    //------------------------------------------------------------------------//
    // Determine if an interlock is raised:                                   //
    //------------------------------------------------------------------------//
    O #tIL.Source[0];
    O #tIL.Source[1];
    O #tIL.Source[2];
    O #tIL.Source[3];
    O #tIL.Source[4];
    O #tIL.Source[5];
    O #tIL.Source[6];
    O #tIL.Source[7];
    O #tIL.Source[8];
    O #tIL.Source[9];
    O #tIL.Source[10];
    O #tIL.Source[11];
    O #tIL.Source[12];
    O #tIL.Source[13];
    O #tIL.Source[14];
    = #tIL.INTERLOCK;

NETWORK
TITLE = Item 77 DV4109 : Update the instance data
    //------------------------------------------------------------------------//
    // Update the instance DB with the calculated interlock flags:            //
    //------------------------------------------------------------------------//
    CALL MOVE
    {value_type := 'Variant'}
    (   IN                   := #tIL ,
        OUT                  := #p[77]
    );

NETWORK
TITLE = Item 78 DV4111 : WFI Supply Valve initialise variables
    //------------------------------------------------------------------------//
    // CRITICAL INTERLOCK   CRITICAL INTERLOCK   CRITICAL INTERLOCK   CRITICA //
    // CRITICAL INTERLOCK   CRITICAL INTERLOCK   CRITICAL INTERLOCK   CRITICA //
    //                                                                        //
    // Clear the interlock flag:                                              //
    //------------------------------------------------------------------------//
    A "alwaysLow";
    = #tIL.INTERLOCK;

    //------------------------------------------------------------------------//
    // Clear all interlock values to initialise them to off:                  //
    //------------------------------------------------------------------------//
    CALL FILL_BLK
    {value_type := 'Bool', count_type := 'UInt'}
    (   IN                   := 0 ,
        COUNT                := 15 ,
        OUT                  := #tIL.Source[0]
    );


NETWORK
TITLE = Item 78 DV4111 interlock source : ON ZSC4107 Vessel inlet line Flowpath Indicator IN   ON ZSC4103 Vessel WFI Supply Flowpath Indicator IN
    //------------------------------------------------------------------------//
    // Calculate the interlock condition:                                     //
    //------------------------------------------------------------------------//
    ON(;
    L "idbZSC2".f[23].p.read.mc.STATE;
    L "dbCONST".BLK.ZSC2.STATE.IN;
    ==I;
    );
ON(;
    L "idbZSC2".f[21].p.read.mc.STATE;
    L "dbCONST".BLK.ZSC2.STATE.IN;
    ==I;
    );
    = #tIL.Source[0];

NETWORK
TITLE = Item 78 DV4111 interlock source : A DV4109 Vessel PS Supply for WFI Loop OPENED
    //------------------------------------------------------------------------//
    // Calculate the interlock condition:                                     //
    //------------------------------------------------------------------------//
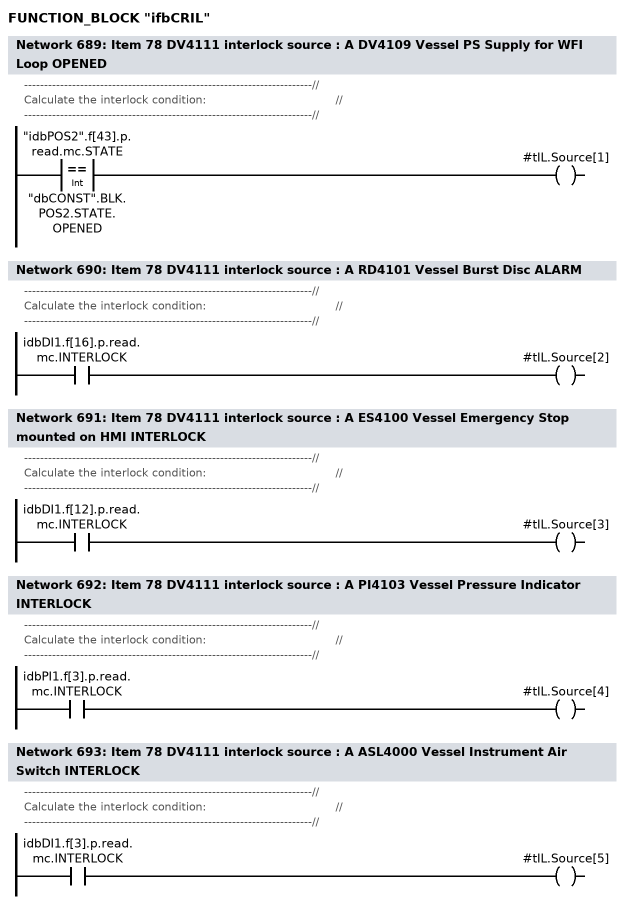
    A(;
    L "idbPOS2".f[43].p.read.mc.STATE;
    L "dbCONST".BLK.POS2.STATE.OPENED;
    ==I;
    );
    = #tIL.Source[1];

NETWORK
TITLE = Item 78 DV4111 interlock source : A RD4101 Vessel Burst Disc ALARM
    //------------------------------------------------------------------------//
    // Calculate the interlock condition:                                     //
    //------------------------------------------------------------------------//
    A idbDI1.f[16].p.read.mc.INTERLOCK;
    = #tIL.Source[2];

NETWORK
TITLE = Item 78 DV4111 interlock source : A ES4100 Vessel Emergency Stop mounted on HMI INTERLOCK
    //------------------------------------------------------------------------//
    // Calculate the interlock condition:                                     //
    //------------------------------------------------------------------------//
    A idbDI1.f[12].p.read.mc.INTERLOCK;
    = #tIL.Source[3];

NETWORK
TITLE = Item 78 DV4111 interlock source : A PI4103 Vessel Pressure Indicator INTERLOCK
    //------------------------------------------------------------------------//
    // Calculate the interlock condition:                                     //
    //------------------------------------------------------------------------//
    A idbPI1.f[3].p.read.mc.INTERLOCK;
    = #tIL.Source[4];

NETWORK
TITLE = Item 78 DV4111 interlock source : A ASL4000 Vessel Instrument Air Switch INTERLOCK
    //------------------------------------------------------------------------//
    // Calculate the interlock condition:                                     //
    //------------------------------------------------------------------------//
    A idbDI1.f[3].p.read.mc.INTERLOCK;
    = #tIL.Source[5];

NETWORK
TITLE = Item 78 DV4111 interlock source : AN ZSC4101 Vessel Manway Closed Indicator CLOSED
    //------------------------------------------------------------------------//
    // Calculate the interlock condition:                                     //
    //------------------------------------------------------------------------//
    AN(;
    L "idbZSC1".f[3].p.read.mc.STATE;
    L "dbCONST".BLK.ZSC1.STATE.CLOSED;
    ==I;
    );
    = #tIL.Source[6];


NETWORK
TITLE = Item 78 DV4111 : Number of interlocks
    //------------------------------------------------------------------------//
    // Number of interlocks
    //------------------------------------------------------------------------//
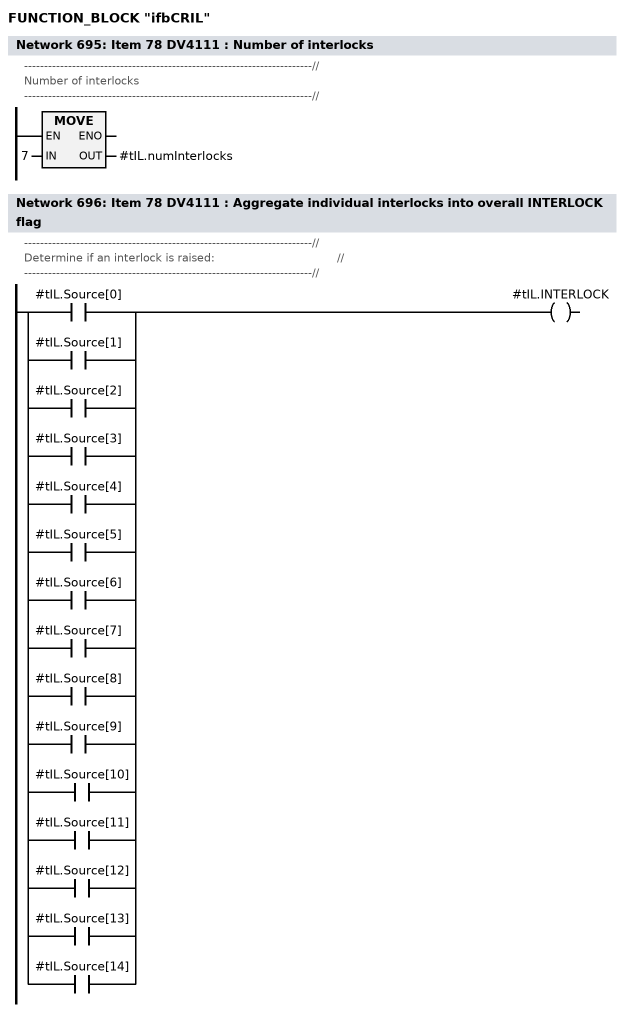
    L 7;
    T #tIL.numInterlocks;

NETWORK
TITLE = Item 78 DV4111 : Aggregate individual interlocks into overall INTERLOCK flag
    //------------------------------------------------------------------------//
    // Determine if an interlock is raised:                                   //
    //------------------------------------------------------------------------//
    O #tIL.Source[0];
    O #tIL.Source[1];
    O #tIL.Source[2];
    O #tIL.Source[3];
    O #tIL.Source[4];
    O #tIL.Source[5];
    O #tIL.Source[6];
    O #tIL.Source[7];
    O #tIL.Source[8];
    O #tIL.Source[9];
    O #tIL.Source[10];
    O #tIL.Source[11];
    O #tIL.Source[12];
    O #tIL.Source[13];
    O #tIL.Source[14];
    = #tIL.INTERLOCK;

NETWORK
TITLE = Item 78 DV4111 : Update the instance data
    //------------------------------------------------------------------------//
    // Update the instance DB with the calculated interlock flags:            //
    //------------------------------------------------------------------------//
    CALL MOVE
    {value_type := 'Variant'}
    (   IN                   := #tIL ,
        OUT                  := #p[78]
    );

NETWORK
TITLE = Item 79 DV4113 : PW Supply Valve initialise variables
    //------------------------------------------------------------------------//
    // CRITICAL INTERLOCK   CRITICAL INTERLOCK   CRITICAL INTERLOCK   CRITICA //
    // CRITICAL INTERLOCK   CRITICAL INTERLOCK   CRITICAL INTERLOCK   CRITICA //
    //                                                                        //
    // Clear the interlock flag:                                              //
    //------------------------------------------------------------------------//
    A "alwaysLow";
    = #tIL.INTERLOCK;

    //------------------------------------------------------------------------//
    // Clear all interlock values to initialise them to off:                  //
    //------------------------------------------------------------------------//
    CALL FILL_BLK
    {value_type := 'Bool', count_type := 'UInt'}
    (   IN                   := 0 ,
        COUNT                := 15 ,
        OUT                  := #tIL.Source[0]
    );


NETWORK
TITLE = Item 79 DV4113 interlock source : ON ZSC4107 Vessel inlet line Flowpath Indicator IN   ON ZSC4105 Vessel PW Supply Flowpath Indicator IN
    //------------------------------------------------------------------------//
    // Calculate the interlock condition:                                     //
    //------------------------------------------------------------------------//
    ON(;
    L "idbZSC2".f[23].p.read.mc.STATE;
    L "dbCONST".BLK.ZSC2.STATE.IN;
    ==I;
    );
ON(;
    L "idbZSC2".f[22].p.read.mc.STATE;
    L "dbCONST".BLK.ZSC2.STATE.IN;
    ==I;
    );
    = #tIL.Source[0];

NETWORK
TITLE = Item 79 DV4113 interlock source : A DV4115 Vessel PS Supply for PW Loop OPENED
    //------------------------------------------------------------------------//
    // Calculate the interlock condition:                                     //
    //------------------------------------------------------------------------//
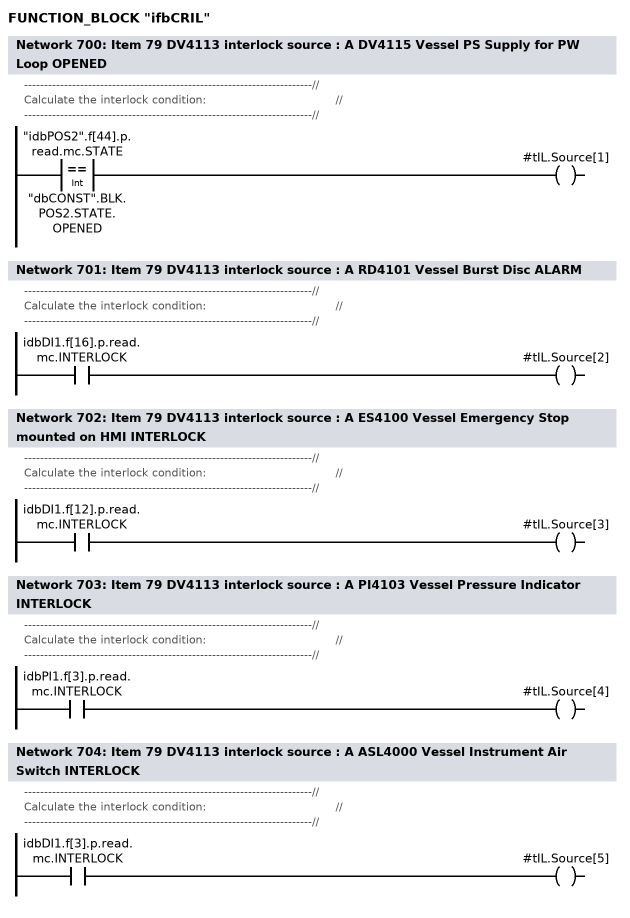
    A(;
    L "idbPOS2".f[44].p.read.mc.STATE;
    L "dbCONST".BLK.POS2.STATE.OPENED;
    ==I;
    );
    = #tIL.Source[1];

NETWORK
TITLE = Item 79 DV4113 interlock source : A RD4101 Vessel Burst Disc ALARM
    //------------------------------------------------------------------------//
    // Calculate the interlock condition:                                     //
    //------------------------------------------------------------------------//
    A idbDI1.f[16].p.read.mc.INTERLOCK;
    = #tIL.Source[2];

NETWORK
TITLE = Item 79 DV4113 interlock source : A ES4100 Vessel Emergency Stop mounted on HMI INTERLOCK
    //------------------------------------------------------------------------//
    // Calculate the interlock condition:                                     //
    //------------------------------------------------------------------------//
    A idbDI1.f[12].p.read.mc.INTERLOCK;
    = #tIL.Source[3];

NETWORK
TITLE = Item 79 DV4113 interlock source : A PI4103 Vessel Pressure Indicator INTERLOCK
    //------------------------------------------------------------------------//
    // Calculate the interlock condition:                                     //
    //------------------------------------------------------------------------//
    A idbPI1.f[3].p.read.mc.INTERLOCK;
    = #tIL.Source[4];

NETWORK
TITLE = Item 79 DV4113 interlock source : A ASL4000 Vessel Instrument Air Switch INTERLOCK
    //------------------------------------------------------------------------//
    // Calculate the interlock condition:                                     //
    //------------------------------------------------------------------------//
    A idbDI1.f[3].p.read.mc.INTERLOCK;
    = #tIL.Source[5];

NETWORK
TITLE = Item 79 DV4113 interlock source : AN ZSC4101 Vessel Manway Closed Indicator CLOSED
    //------------------------------------------------------------------------//
    // Calculate the interlock condition:                                     //
    //------------------------------------------------------------------------//
    AN(;
    L "idbZSC1".f[3].p.read.mc.STATE;
    L "dbCONST".BLK.ZSC1.STATE.CLOSED;
    ==I;
    );
    = #tIL.Source[6];


NETWORK
TITLE = Item 79 DV4113 : Number of interlocks
    //------------------------------------------------------------------------//
    // Number of interlocks
    //------------------------------------------------------------------------//
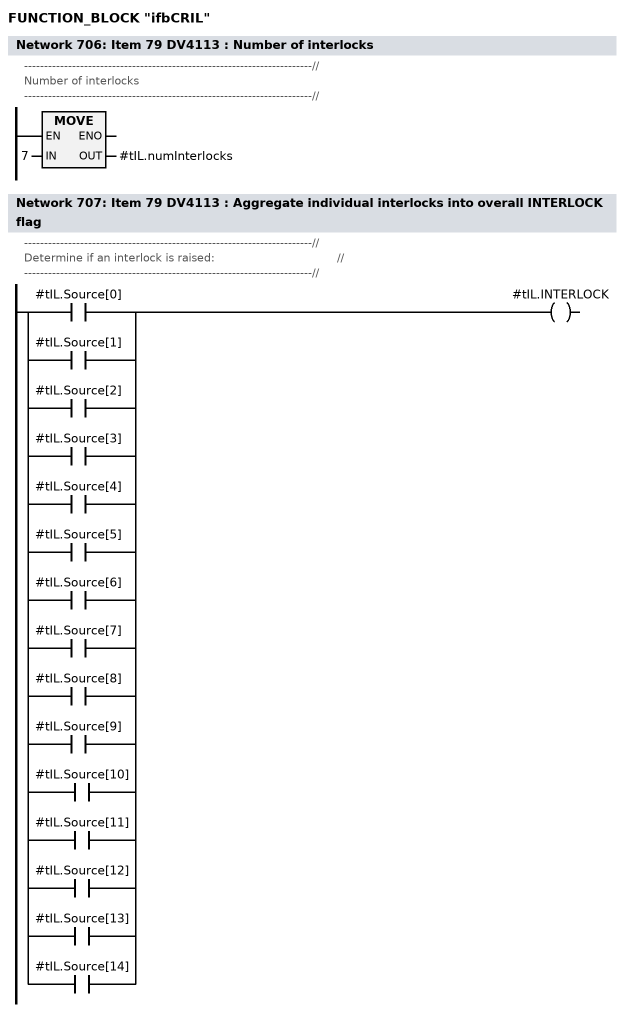
    L 7;
    T #tIL.numInterlocks;

NETWORK
TITLE = Item 79 DV4113 : Aggregate individual interlocks into overall INTERLOCK flag
    //------------------------------------------------------------------------//
    // Determine if an interlock is raised:                                   //
    //------------------------------------------------------------------------//
    O #tIL.Source[0];
    O #tIL.Source[1];
    O #tIL.Source[2];
    O #tIL.Source[3];
    O #tIL.Source[4];
    O #tIL.Source[5];
    O #tIL.Source[6];
    O #tIL.Source[7];
    O #tIL.Source[8];
    O #tIL.Source[9];
    O #tIL.Source[10];
    O #tIL.Source[11];
    O #tIL.Source[12];
    O #tIL.Source[13];
    O #tIL.Source[14];
    = #tIL.INTERLOCK;

NETWORK
TITLE = Item 79 DV4113 : Update the instance data
    //------------------------------------------------------------------------//
    // Update the instance DB with the calculated interlock flags:            //
    //------------------------------------------------------------------------//
    CALL MOVE
    {value_type := 'Variant'}
    (   IN                   := #tIL ,
        OUT                  := #p[79]
    );

NETWORK
TITLE = Item 80 DV4115 : PS Supply for PW Loop initialise variables
    //------------------------------------------------------------------------//
    // CRITICAL INTERLOCK   CRITICAL INTERLOCK   CRITICAL INTERLOCK   CRITICA //
    // CRITICAL INTERLOCK   CRITICAL INTERLOCK   CRITICAL INTERLOCK   CRITICA //
    //                                                                        //
    // Clear the interlock flag:                                              //
    //------------------------------------------------------------------------//
    A "alwaysLow";
    = #tIL.INTERLOCK;

    //------------------------------------------------------------------------//
    // Clear all interlock values to initialise them to off:                  //
    //------------------------------------------------------------------------//
    CALL FILL_BLK
    {value_type := 'Bool', count_type := 'UInt'}
    (   IN                   := 0 ,
        COUNT                := 15 ,
        OUT                  := #tIL.Source[0]
    );


NETWORK
TITLE = Item 80 DV4115 interlock source : ON ZSC4107 Vessel inlet line Flowpath Indicator IN   ON ZSC4105 Vessel PW Supply Flowpath Indicator IN
    //------------------------------------------------------------------------//
    // Calculate the interlock condition:                                     //
    //------------------------------------------------------------------------//
    ON(;
    L "idbZSC2".f[23].p.read.mc.STATE;
    L "dbCONST".BLK.ZSC2.STATE.IN;
    ==I;
    );
ON(;
    L "idbZSC2".f[22].p.read.mc.STATE;
    L "dbCONST".BLK.ZSC2.STATE.IN;
    ==I;
    );
    = #tIL.Source[0];

NETWORK
TITLE = Item 80 DV4115 interlock source : A DV4113 Vessel PW Supply Valve OPENED
    //------------------------------------------------------------------------//
    // Calculate the interlock condition:                                     //
    //------------------------------------------------------------------------//
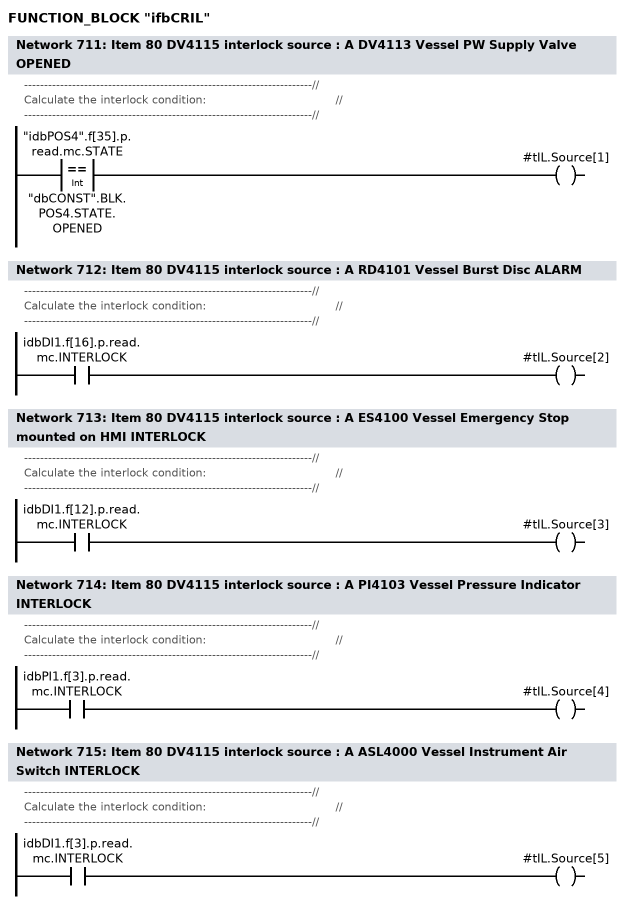
    A(;
    L "idbPOS4".f[35].p.read.mc.STATE;
    L "dbCONST".BLK.POS4.STATE.OPENED;
    ==I;
    );
    = #tIL.Source[1];

NETWORK
TITLE = Item 80 DV4115 interlock source : A RD4101 Vessel Burst Disc ALARM
    //------------------------------------------------------------------------//
    // Calculate the interlock condition:                                     //
    //------------------------------------------------------------------------//
    A idbDI1.f[16].p.read.mc.INTERLOCK;
    = #tIL.Source[2];

NETWORK
TITLE = Item 80 DV4115 interlock source : A ES4100 Vessel Emergency Stop mounted on HMI INTERLOCK
    //------------------------------------------------------------------------//
    // Calculate the interlock condition:                                     //
    //------------------------------------------------------------------------//
    A idbDI1.f[12].p.read.mc.INTERLOCK;
    = #tIL.Source[3];

NETWORK
TITLE = Item 80 DV4115 interlock source : A PI4103 Vessel Pressure Indicator INTERLOCK
    //------------------------------------------------------------------------//
    // Calculate the interlock condition:                                     //
    //------------------------------------------------------------------------//
    A idbPI1.f[3].p.read.mc.INTERLOCK;
    = #tIL.Source[4];

NETWORK
TITLE = Item 80 DV4115 interlock source : A ASL4000 Vessel Instrument Air Switch INTERLOCK
    //------------------------------------------------------------------------//
    // Calculate the interlock condition:                                     //
    //------------------------------------------------------------------------//
    A idbDI1.f[3].p.read.mc.INTERLOCK;
    = #tIL.Source[5];

NETWORK
TITLE = Item 80 DV4115 interlock source : AN ZSC4101 Vessel Manway Closed Indicator CLOSED
    //------------------------------------------------------------------------//
    // Calculate the interlock condition:                                     //
    //------------------------------------------------------------------------//
    AN(;
    L "idbZSC1".f[3].p.read.mc.STATE;
    L "dbCONST".BLK.ZSC1.STATE.CLOSED;
    ==I;
    );
    = #tIL.Source[6];


NETWORK
TITLE = Item 80 DV4115 : Number of interlocks
    //------------------------------------------------------------------------//
    // Number of interlocks
    //------------------------------------------------------------------------//
